Staubli VAL3: parseMovement.pgx

program parseMovement()
begin
  //putln(sInput)
  sGetMovement=sInput[0]

  sGetMovement=toNum(sGetMovement,nXMovement,bParseResult)
  sGetMovement=toNum(sGetMovement,nZMovement,bParseResult)
  sGetMovement=toNum(sGetMovement,nRXMovement,bParseResult)

  //putln(nXMovement)
  //putln(nZMovement)
  //putln(nRXMovement)

  call actMovement()
end
